# EPICS substitutions: vacuum/MAIN_TRUNK/vacApp/Db/dc1_agilent4uhv.substitutions
# Agilent4UHV substitutions file

file db/agilent4uhv.db
{
     pattern {LOCA,			DEV,		PORT,		ADDR,	TIMEOUT}
     		 {SL3,			DC1,		4uhv_1,		0,		0.2}
}
file db/agilent4uhv_alias.db
{
     pattern {LOCA,			DEV,		SUB1,					SUB2,					SUB3,						SUB4,				PORT,	ADDR,	TIMEOUT}
     		 {SL3,			DC1,	Empty,		VDR:IP02:SIP30,		VDR:IP03:SIP30,			VDR:IP04:IP30,	4uhv_1,	0,		0.2}
}
